FUNCTION_BLOCK xPlanarMovements
VAR_INPUT
END_VAR
VAR_OUTPUT
END_VAR
VAR
	Running			: BYTE;
	i				: BYTE;
	MainState		: BYTE;
	State			: BYTE;
	
	MoveParameters	: ARRAY [1..xPlanarLink.MoverCount] OF ST_MoverParameters;
	
	EndTimer		: TON;
	MidTimer		: TON;
	
	StartSequence	: BOOL;
	CommandDone		: BOOL;
	MoveDone		: BOOL;
	
	Velocity		: LREAL := 2000;
END_VAR

METHOD PUBLIC DecreaseMoverHeight : BOOL
VAR_INPUT
	Run		: BOOL;
END_VAR

// Movers go a bit low

IF Run THEN

	MoveDone := FALSE;
	
	CASE State OF
		
		0:
			State := 1;
	
		
		1:
			FOR i := 1 TO xPlanarLink.MoverCount DO
				xPlanarLink.PlanarMover[i].MoveZ
				(	
					commandFeedback		:= xPlanarLink.PlanarFeedback[i],
					targetPosition		:= 2.0,
					constraint			:= MoveParameters[i].Constraints
				);
			END_FOR
			State := 2;
		
		2:
			CommandDone := xPlanarLink.PlanarFeedback[1].Done AND xPlanarLink.PlanarFeedback[2].Done;
			
			IF CommandDone THEN
				CommandDone := FALSE;
				State := 3;
			END_IF
	
		3:
			MoveDone := TRUE;
			State := 0;
	
	END_CASE

END_IF
END_METHOD

METHOD DefineParameters : BOOL
VAR_INPUT
END_VAR

// Define the movement parameters for this demo

MoveParameters[1].Options.useOrientation := TRUE;
MoveParameters[1].Constraints.SetValuesVADJ(V := Velocity, A := 20000, D := 20000, J := 200000);
MoveParameters[1].rotateOptions.additionalTurns := 5;
MoveParameters[1].rotateOptions.direction := 1;

MoveParameters[2].Options.useOrientation := TRUE;
MoveParameters[2].Constraints.SetValuesVADJ(V := Velocity, A := 20000, D := 20000, J := 200000);
MoveParameters[2].rotateOptions.additionalTurns := 5;
MoveParameters[2].rotateOptions.direction := 3;
END_METHOD

METHOD DelayBetweenMoves : BOOL
VAR_INPUT
	Start		: BOOL;
	Delay		: TIME;
END_VAR

MoveDone := FALSE;

MidTimer(IN := Start, PT := Delay);

IF MidTimer.Q THEN
	MoveDone := TRUE;
END_IF
END_METHOD

METHOD EndDelay : BOOL
VAR_INPUT
	Start		: BOOL;
	Delay		: TIME;
END_VAR

MoveDone := FALSE;

EndTimer(IN := Start, PT := Delay);

IF EndTimer.Q THEN
	MoveDone := TRUE;
END_IF
END_METHOD

METHOD PUBLIC FollowTileEdge : BOOL
VAR_INPUT
	Run		: BOOL;
END_VAR

// Movers move to edge of tiles and follow the perimeter, then move to home

IF Run THEN

	MoveDone := FALSE;
	
	CASE State OF
		
		0:
			State := 1;
	
		1:
			MoveParameters[1].targetPosition.x := 180;
			MoveParameters[1].targetPosition.y := 183;
			MoveParameters[2].targetPosition.x := 296;
			MoveParameters[2].targetPosition.y := 183;
			State := 2;
		
		2:
			FOR i := 1 TO xPlanarLink.MoverCount DO
				xPlanarLink.PlanarMover[i].MoveToPosition
				(
					commandFeedback 	:= xPlanarLink.PlanarFeedback[i],
					targetPosition 		:= MoveParameters[i].targetPosition,
					constraint 			:= MoveParameters[i].Constraints,
					options 			:= MoveParameters[i].Options
				);
			END_FOR
			State := 3;
		
		3:
			FOR i := 1 TO xPlanarLink.MoverCount DO
				CommandDone := xPlanarLink.PlanarFeedback[i].Done;
			END_FOR
			
			IF CommandDone THEN
				CommandDone := FALSE;
				State := 4;
			END_IF
	
		4:
			moveParameters[1].targetPosition.x := 57;
			moveParameters[1].targetPosition.y := 183;
			moveParameters[2].targetPosition.x := 423;
			moveParameters[2].targetPosition.y := 183;
			State := 5;
		
		5:
			FOR i := 1 TO xPlanarLink.MoverCount DO
				xPlanarLink.PlanarMover[i].MoveToPosition
				(
					commandFeedback 	:= xPlanarLink.PlanarFeedback[i],
					targetPosition 		:= MoveParameters[i].targetPosition,
					constraint 			:= MoveParameters[i].Constraints,
					options 			:= MoveParameters[i].Options
				);
			END_FOR
			State := 6;
		
		6:
			FOR i := 1 TO xPlanarLink.MoverCount DO
				CommandDone := xPlanarLink.PlanarFeedback[i].Done;
			END_FOR
			
			IF CommandDone THEN
				CommandDone := FALSE;
				State := 7;
			END_IF
			
		7:
			moveParameters[1].targetPosition.x := 57;
			moveParameters[1].targetPosition.y := 57;
			moveParameters[2].targetPosition.x := 423;
			moveParameters[2].targetPosition.y := 57;
			State := 8;
		
		8:
			FOR i := 1 TO xPlanarLink.MoverCount DO
				xPlanarLink.PlanarMover[i].MoveToPosition
				(
					commandFeedback 	:= xPlanarLink.PlanarFeedback[i],
					targetPosition 		:= MoveParameters[i].targetPosition,
					constraint 			:= MoveParameters[i].Constraints,
					options 			:= MoveParameters[i].Options
				);
			END_FOR
			State := 9;
		
		9:
			FOR i := 1 TO xPlanarLink.MoverCount DO
				CommandDone := xPlanarLink.PlanarFeedback[i].Done;
			END_FOR
			
			IF CommandDone THEN
				CommandDone := FALSE;
				State := 10;
			END_IF
			
		10:
			moveParameters[1].targetPosition.x := 180;
			moveParameters[1].targetPosition.y := 57;
			moveParameters[2].targetPosition.x := 296;
			moveParameters[2].targetPosition.y := 57;
			State := 11;
		
		11:
			FOR i := 1 TO xPlanarLink.MoverCount DO
				xPlanarLink.PlanarMover[i].MoveToPosition
				(
					commandFeedback 	:= xPlanarLink.PlanarFeedback[i],
					targetPosition 		:= MoveParameters[i].targetPosition,
					constraint 			:= MoveParameters[i].Constraints,
					options 			:= MoveParameters[i].Options
				);
			END_FOR
			State := 12;
		
		12:
			FOR i := 1 TO xPlanarLink.MoverCount DO
				CommandDone := xPlanarLink.PlanarFeedback[i].Done;
			END_FOR
			
			IF CommandDone THEN
				CommandDone := FALSE;
				State := 13;
			END_IF
			
		13:
			moveParameters[1].targetPosition.x := 120;
			moveParameters[1].targetPosition.y := 120;
			moveParameters[2].targetPosition.x := 360;
			moveParameters[2].targetPosition.y := 120;
			State := 14;
		
		14:
			FOR i := 1 TO xPlanarLink.MoverCount DO
				xPlanarLink.PlanarMover[i].MoveToPosition
				(
					commandFeedback 	:= xPlanarLink.PlanarFeedback[i],
					targetPosition 		:= MoveParameters[i].targetPosition,
					constraint 			:= MoveParameters[i].Constraints,
					options 			:= MoveParameters[i].Options
				);
			END_FOR
			State := 15;
		
		15:
			FOR i := 1 TO xPlanarLink.MoverCount DO
				CommandDone := xPlanarLink.PlanarFeedback[i].Done;
			END_FOR
			
			IF CommandDone THEN
				CommandDone := FALSE;
				State := 16;
			END_IF
			
		16:
			MoveDone := TRUE;
			State := 0;
			
	END_CASE		

END_IF
END_METHOD

METHOD PUBLIC Home : BOOL
VAR_INPUT
	Run		: BOOL;
END_VAR

// Move movers to the middle of tiles.
IF Run THEN

	MoveDone := FALSE;
	
	CASE State OF
			
		0:
			State := 1;
			
		1:
			moveParameters[1].targetPosition.x := 120;
			moveParameters[1].targetPosition.y := 120;
			moveParameters[2].targetPosition.x := 360;
			moveParameters[2].targetPosition.y := 120;
			State := 2;
			
		2:
			FOR i := 1 TO xPlanarLink.MoverCount DO
				xPlanarLink.PlanarMover[i].MoveToPosition
				(
					commandFeedback 	:= xPlanarLink.PlanarFeedback[i],
					targetPosition 		:= MoveParameters[i].targetPosition,
					constraint 			:= MoveParameters[i].Constraints,
					options 			:= MoveParameters[i].Options
				);
			END_FOR
			State := 3;
			
		3:
			CommandDone := xPlanarLink.PlanarFeedback[1].Done AND xPlanarLink.PlanarFeedback[2].Done;
			
			IF CommandDone THEN
				CommandDone := FALSE;
				State := 4;
			END_IF
			
		4:
			MoveDone := TRUE;
			State := 0;
			
			
	END_CASE

END_IF
END_METHOD

METHOD PUBLIC Spin : BOOL
VAR_INPUT
	Run		: BOOL;
END_VAR




// Movers spin

IF Run THEN
	
	MoveDone := FALSE;
	
	CASE State OF
		
		0:
			State := 1;
	
		
		1:
			FOR i := 1 TO xPlanarLink.MoverCount DO
				xPlanarLink.PlanarMover[i].MoveC
				(	
					commandFeedback		:= xPlanarLink.PlanarFeedback[i],
					targetPosition		:= 0,
					constraint			:= MoveParameters[i].Constraints,
					options 			:= MoveParameters[i].rotateOptions
				);
			END_FOR
			State := 2;
		
		2:
			CommandDone := xPlanarLink.PlanarFeedback[1].Done AND xPlanarLink.PlanarFeedback[2].Done;
			
			IF CommandDone THEN
				CommandDone := FALSE;
				State := 3;
			END_IF
			
		3:
			MoveDone := TRUE;
			State := 0;
		
	END_CASE
	
END_IF
END_METHOD

METHOD PUBLIC SwapPlaces : BOOL
VAR_INPUT
	Run		: BOOL;
END_VAR

// Movers swap tiles, then swap back, then move to home

IF Run THEN
	
	MoveDone := FALSE;
	
	CASE State OF
		
		0:
			State := 1;
	
		1:
			MoveParameters[1].targetPosition.x := 175;
			MoveParameters[1].targetPosition.y := 183;
			MoveParameters[2].targetPosition.x := 301;
			MoveParameters[2].targetPosition.y := 57;
			State := 2;
		
		2:
			FOR i := 1 TO xPlanarLink.MoverCount DO
				xPlanarLink.PlanarMover[i].MoveToPosition
				(
					commandFeedback 	:= xPlanarLink.PlanarFeedback[i],
					targetPosition 		:= MoveParameters[i].targetPosition,
					constraint 			:= MoveParameters[i].Constraints,
					options 			:= MoveParameters[i].Options
				);
			END_FOR
			State := 3;
		
		3:
			CommandDone := xPlanarLink.PlanarFeedback[1].Done AND xPlanarLink.PlanarFeedback[2].Done;
			
			IF CommandDone THEN
				CommandDone := FALSE;
				State := 4;
			END_IF
	
		4:
			moveParameters[1].targetPosition.x := 301;
			moveParameters[1].targetPosition.y := 183;
			moveParameters[2].targetPosition.x := 175;
			moveParameters[2].targetPosition.y := 57;
			State := 5;
		
		5:
			FOR i := 1 TO xPlanarLink.MoverCount DO
				xPlanarLink.PlanarMover[i].MoveToPosition
				(
					commandFeedback 	:= xPlanarLink.PlanarFeedback[i],
					targetPosition 		:= MoveParameters[i].targetPosition,
					constraint 			:= MoveParameters[i].Constraints,
					options 			:= MoveParameters[i].Options
				);
			END_FOR
			State := 6;
		
		6:
			CommandDone := xPlanarLink.PlanarFeedback[1].Done AND xPlanarLink.PlanarFeedback[2].Done;
			
			IF CommandDone THEN
				CommandDone := FALSE;
				State := 7;
			END_IF
			
		7:
			moveParameters[1].targetPosition.x := 301;
			moveParameters[1].targetPosition.y := 57;
			moveParameters[2].targetPosition.x := 175;
			moveParameters[2].targetPosition.y := 183;
			State := 8;
		
		8:
			FOR i := 1 TO xPlanarLink.MoverCount DO
				xPlanarLink.PlanarMover[i].MoveToPosition
				(
					commandFeedback 	:= xPlanarLink.PlanarFeedback[i],
					targetPosition 		:= MoveParameters[i].targetPosition,
					constraint 			:= MoveParameters[i].Constraints,
					options 			:= MoveParameters[i].Options
				);
			END_FOR
			State := 9;
		
		9:
			CommandDone := xPlanarLink.PlanarFeedback[1].Done AND xPlanarLink.PlanarFeedback[2].Done;
			
			IF CommandDone THEN
				CommandDone := FALSE;
				State := 10;
			END_IF
			
		10:
			moveParameters[1].targetPosition.x := 175;
			moveParameters[1].targetPosition.y := 57;
			moveParameters[2].targetPosition.x := 301;
			moveParameters[2].targetPosition.y := 183;
			State := 11;
		
		11:
			FOR i := 1 TO xPlanarLink.MoverCount DO
				xPlanarLink.PlanarMover[i].MoveToPosition
				(
					commandFeedback 	:= xPlanarLink.PlanarFeedback[i],
					targetPosition 		:= MoveParameters[i].targetPosition,
					constraint 			:= MoveParameters[i].Constraints,
					options 			:= MoveParameters[i].Options
				);
			END_FOR
			State := 12;
		
		12:
			CommandDone := xPlanarLink.PlanarFeedback[1].Done AND xPlanarLink.PlanarFeedback[2].Done;
			
			IF CommandDone THEN
				CommandDone := FALSE;
				State := 13;
			END_IF
			
		13:
			moveParameters[1].targetPosition.x := 120;
			moveParameters[1].targetPosition.y := 120;
			moveParameters[2].targetPosition.x := 360;
			moveParameters[2].targetPosition.y := 120;
			State := 14;
		
		14:
			FOR i := 1 TO xPlanarLink.MoverCount DO
				xPlanarLink.PlanarMover[i].MoveToPosition
				(
					commandFeedback 	:= xPlanarLink.PlanarFeedback[i],
					targetPosition 		:= MoveParameters[i].targetPosition,
					constraint 			:= MoveParameters[i].Constraints,
					options 			:= MoveParameters[i].Options
				);
			END_FOR
			State := 15;
		
		15:
			CommandDone := xPlanarLink.PlanarFeedback[1].Done AND xPlanarLink.PlanarFeedback[2].Done;
			
			IF CommandDone THEN
				CommandDone := FALSE;
				State := 16;
			END_IF
			
		16:
			MoveDone := TRUE;
			State := 0;
			
	END_CASE		
	
END_IF
END_METHOD

METHOD PUBLIC Tilt : BOOL
VAR_INPUT
	Run		: BOOL;
END_VAR

// Movers tilt

IF Run THEN
	
	MoveDone := FALSE;
	
	CASE State OF
		
		0:
			State := 1;
			
		1:
			FOR i := 1 TO xPlanarLink.MoverCount DO
				xPlanarLink.PlanarMover[i].MoveZ
				(	
					commandFeedback		:= xPlanarLink.PlanarFeedback[i],
					targetPosition		:= 5.0,
					constraint			:= MoveParameters[i].Constraints
				);
			END_FOR
			State := 2;
		
		2:
			CommandDone := xPlanarLink.PlanarFeedback[1].Done AND xPlanarLink.PlanarFeedback[2].Done;
			
			IF CommandDone THEN
				CommandDone := FALSE;
				State := 3;
			END_IF
	
		
		3:
			FOR i := 1 TO xPlanarLink.MoverCount DO
				xPlanarLink.PlanarMover[i].MoveA
				(	
					commandFeedback		:= xPlanarLink.PlanarFeedback[i],
					targetPosition		:= 4.0,
					constraint			:= MoveParameters[i].Constraints
				);
			END_FOR
			State := 4;
		
		4:
			CommandDone := xPlanarLink.PlanarFeedback[1].Done AND xPlanarLink.PlanarFeedback[2].Done;
			
			IF CommandDone THEN
				CommandDone := FALSE;
				State := 5;
			END_IF
			
		5:
			FOR i := 1 TO xPlanarLink.MoverCount DO
				xPlanarLink.PlanarMover[i].MoveA
				(	
					commandFeedback		:= xPlanarLink.PlanarFeedback[i],
					targetPosition		:= -4.0,
					constraint			:= MoveParameters[i].Constraints
				);
			END_FOR
			State := 6;
		
		6:
			CommandDone := xPlanarLink.PlanarFeedback[1].Done AND xPlanarLink.PlanarFeedback[2].Done;
			
			IF CommandDone THEN
				CommandDone := FALSE;
				State := 7;
			END_IF
		
		7:
			FOR i := 1 TO xPlanarLink.MoverCount DO
				xPlanarLink.PlanarMover[i].MoveA
				(	
					commandFeedback		:= xPlanarLink.PlanarFeedback[i],
					targetPosition		:= 0.0,
					constraint			:= MoveParameters[i].Constraints
				);
			END_FOR
			State := 8;
		
		8:
			CommandDone := xPlanarLink.PlanarFeedback[1].Done AND xPlanarLink.PlanarFeedback[2].Done;
			
			IF CommandDone THEN
				CommandDone := FALSE;
				State := 9;
			END_IF
			
		9:
			FOR i := 1 TO xPlanarLink.MoverCount DO
				xPlanarLink.PlanarMover[i].MoveB
				(	
					commandFeedback		:= xPlanarLink.PlanarFeedback[i],
					targetPosition		:= 4.0,
					constraint			:= MoveParameters[i].Constraints
				);
			END_FOR
			State := 10;
		
		10:
			CommandDone := xPlanarLink.PlanarFeedback[1].Done AND xPlanarLink.PlanarFeedback[2].Done;
			
			IF CommandDone THEN
				CommandDone := FALSE;
				State := 11;
			END_IF
			
		11:
			FOR i := 1 TO xPlanarLink.MoverCount DO
				xPlanarLink.PlanarMover[i].MoveB
				(	
					commandFeedback		:= xPlanarLink.PlanarFeedback[i],
					targetPosition		:= -4.0,
					constraint			:= MoveParameters[i].Constraints
				);
			END_FOR
			State := 12;
		
		12:
			CommandDone := xPlanarLink.PlanarFeedback[1].Done AND xPlanarLink.PlanarFeedback[2].Done;
			
			IF CommandDone THEN
				CommandDone := FALSE;
				State := 13;
			END_IF
		
		13:
			FOR i := 1 TO xPlanarLink.MoverCount DO
				xPlanarLink.PlanarMover[i].MoveB
				(	
					commandFeedback		:= xPlanarLink.PlanarFeedback[i],
					targetPosition		:= 0.0,
					constraint			:= MoveParameters[i].Constraints
				);
			END_FOR
			State := 14;
		
		14:
			CommandDone := xPlanarLink.PlanarFeedback[1].Done AND xPlanarLink.PlanarFeedback[2].Done;
			
			IF CommandDone THEN
				CommandDone := FALSE;
				State := 15;
			END_IF
			
		15:
			FOR i := 1 TO xPlanarLink.MoverCount DO
				xPlanarLink.PlanarMover[i].MoveZ
				(	
					commandFeedback		:= xPlanarLink.PlanarFeedback[i],
					targetPosition		:= 2.0,
					constraint			:= MoveParameters[i].Constraints
				);
			END_FOR
			State := 16;
		
		16:
			CommandDone := xPlanarLink.PlanarFeedback[1].Done AND xPlanarLink.PlanarFeedback[2].Done;
			
			IF CommandDone THEN
				CommandDone := FALSE;
				State := 17;
			END_IF
			
		17:
			MoveDone := TRUE;
			State := 0;
			
		
	END_CASE
	
END_IF
END_METHOD

METHOD PUBLIC VaryMoverHeight : BOOL
VAR_INPUT
	Run		: BOOL;
END_VAR

// Movers go a bit high

IF Run THEN
	
	MoveDone := FALSE;
	
	CASE State OF
		
		0:
			State := 1;
	
		
		1:
			FOR i := 1 TO xPlanarLink.MoverCount DO
				xPlanarLink.PlanarMover[i].MoveZ
				(	
					commandFeedback		:= xPlanarLink.PlanarFeedback[i],
					targetPosition		:= 5.0,
					constraint			:= MoveParameters[i].Constraints
				);
			END_FOR
			State := 2;
		
		2:
			CommandDone := xPlanarLink.PlanarFeedback[1].Done AND xPlanarLink.PlanarFeedback[2].Done;
			
			IF CommandDone THEN
				CommandDone := FALSE;
				State := 3;
			END_IF
			
		3:
			FOR i := 1 TO xPlanarLink.MoverCount DO
				xPlanarLink.PlanarMover[i].MoveZ
				(	
					commandFeedback		:= xPlanarLink.PlanarFeedback[i],
					targetPosition		:= 2.0,
					constraint			:= MoveParameters[i].Constraints
				);
			END_FOR
			State := 4;
		
		4:
			CommandDone := xPlanarLink.PlanarFeedback[1].Done AND xPlanarLink.PlanarFeedback[2].Done;
			
			IF CommandDone THEN
				CommandDone := FALSE;
				State := 5;
			END_IF
			
		5:
			FOR i := 1 TO xPlanarLink.MoverCount DO
				xPlanarLink.PlanarMover[i].MoveZ
				(	
					commandFeedback		:= xPlanarLink.PlanarFeedback[i],
					targetPosition		:= 5.0,
					constraint			:= MoveParameters[i].Constraints
				);
			END_FOR
			State := 6;
		
		6:
			CommandDone := xPlanarLink.PlanarFeedback[1].Done AND xPlanarLink.PlanarFeedback[2].Done;
			
			IF CommandDone THEN
				CommandDone := FALSE;
				State := 7;
			END_IF
			
		7:
			FOR i := 1 TO xPlanarLink.MoverCount DO
				xPlanarLink.PlanarMover[i].MoveZ
				(	
					commandFeedback		:= xPlanarLink.PlanarFeedback[i],
					targetPosition		:= 2.0,
					constraint			:= MoveParameters[i].Constraints
				);
			END_FOR
			State := 8;
		
		8:
			CommandDone := xPlanarLink.PlanarFeedback[1].Done AND xPlanarLink.PlanarFeedback[2].Done;
			
			IF CommandDone THEN
				CommandDone := FALSE;
				State := 9;
			END_IF
			
		9:
			FOR i := 1 TO xPlanarLink.MoverCount DO
				xPlanarLink.PlanarMover[i].MoveZ
				(	
					commandFeedback		:= xPlanarLink.PlanarFeedback[i],
					targetPosition		:= 5.0,
					constraint			:= MoveParameters[i].Constraints
				);
			END_FOR
			State := 10;
		
		10:
			CommandDone := xPlanarLink.PlanarFeedback[1].Done AND xPlanarLink.PlanarFeedback[2].Done;
			
			IF CommandDone THEN
				CommandDone := FALSE;
				State := 11;
			END_IF
	
		11:
			FOR i := 1 TO xPlanarLink.MoverCount DO
				xPlanarLink.PlanarMover[i].MoveZ
				(	
					commandFeedback		:= xPlanarLink.PlanarFeedback[i],
					targetPosition		:= 2.0,
					constraint			:= MoveParameters[i].Constraints
				);
			END_FOR
			State := 12;
		
		12:
			CommandDone := xPlanarLink.PlanarFeedback[1].Done AND xPlanarLink.PlanarFeedback[2].Done;
			
			IF CommandDone THEN
				CommandDone := FALSE;
				State := 13;
			END_IF
			
		13:
			MoveDone := TRUE;
			State := 0;
	
	END_CASE
	
END_IF
END_METHOD

END_FUNCTION_BLOCK

(* stored: Version 1.1.0.1, ProductVersion 3.1.4024.12
   POU xPlanarMovements: Id {61237aaa-fa06-4339-bbeb-d7ee6e21aecc}, SpecialFunc None
   Method DecreaseMoverHeight: Id {b14d889b-19a0-45d9-a416-bc5f9f09ddd4}
   Method DefineParameters: Id {e0aafccf-9e5d-40fc-89f7-7cde95b1d36f}
   Method DelayBetweenMoves: Id {75868d57-7e3a-4bf5-96ba-8ac467e4a3b3}
   Method EndDelay: Id {8a494a48-74fe-48d2-9bf0-974a9c61f4ff}
   Method FollowTileEdge: Id {d6a47a68-e1e2-4f06-a26f-1c1effc568f1}
   Method Home: Id {d2cf8f88-7414-44ed-bbfa-414960b0aded}
   Method Spin: Id {5209d939-b863-4f1c-b951-9ae97fddb209}
   Method SwapPlaces: Id {5134322d-04a7-4bd7-abf6-69c5d4a51d36}
   Method Tilt: Id {4ecde7e2-fe03-4893-8dad-a4278fecb2b2}
   Method VaryMoverHeight: Id {ab0c66ae-7e12-4764-9704-cca2fb9445e1} *)
